(* PLC project , Schneider Electric EcoStruxure Machine Expert *)

PROGRAM Main

PROGRAM Main
VAR
    Ready : BOOL := TRUE;
END_VAR
END_PROGRAM
END_PROGRAM

PROGRAM MotorFb

END_PROGRAM
